// TwinCAT 3 PLC project MotionPractise
// ProgramVersion: 3.1.4023.0
// libraries:
//   Tc2_MC2, * (Beckhoff Automation GmbH)
//   Tc2_Standard, * (Beckhoff Automation GmbH)
//   Tc2_System, * (Beckhoff Automation GmbH)
//   Tc3_Module, * (Beckhoff Automation GmbH)
// project tree:
//   / PlcTask.TcTTO
//   POUs/AxisInterface/ Global_Axif_Const.TcGVL, Global_Axis_Interface.TcGVL, TE_AxisBasic_V2.TcPOU, TE_AxisInterface_type01.TcPOU
//   POUs/AxisInterface/Type/ Axis_Ctrl_gb.TcDUT, Axis_Status_gb.TcDUT, E_MotorDirection.TcDUT
//   POUs/AxisInterface/Type/Control/ E_AXIS_MODE.TcDUT, ST_AXIS_ADMINISTRATION.TcDUT, ST_AXIS_MODE_BITS.TcDUT, ST_AXIS_POSITION.TcDUT, ST_AXIS_SETUP_MODE.TcDUT, ST_AXIS_SYNCHRONISATION.TcDUT, ST_AXIS_TORQUE.TcDUT, ST_AXIS_VELOCITY.TcDUT, U_AXIS_MODE.TcDUT
//   POUs/AxisInterface/Type/Status/ ST_AXIS_ADMIN_STATUS.TcDUT, ST_AXIS_DIAGNOSIS.TcDUT, ST_AXIS_POS_STATUS.TcDUT, ST_AXIS_SETUP_MODE_STATUS.TcDUT, ST_AXIS_SYNC_STATUS.TcDUT, ST_AXIS_VEL_STATUS.TcDUT
//   POUs/ MAIN.TcPOU
// real-time tasks:
//   TASK PlcTask: cycle T#10ms, priority 20, ADS port 350
// motion (NC):
//   TASK NC-Task 1 SAF: cycle T#2ms, priority 4, ADS port 501
//   TASK NC-Task 1 SVB: cycle T#10ms, priority 8, ADS port 511
//   AXIS Axis 1 (id 1)
//     OtherSettings: AllowMotionCmdToSlave=true
//     encoder EncType=1
//     drive DrvType=5
//       Analog: TorqueSetpointScale=10, ScaleFactorActTorque=0.1
//     controller CtrType=1
//       CtrPara: PriorControlFactor=1
//         Observer: BandWidth=20
//   AXIS Axis 2 (id 2)
//     OtherSettings: AllowMotionCmdToSlave=true
//     encoder EncType=1
//     drive DrvType=5
//       Analog: TorqueSetpointScale=10, ScaleFactorActTorque=0.1
//     controller CtrType=1
//       CtrPara: PriorControlFactor=1
//         Observer: BandWidth=20
// variable links:
//   MotionPractise/MotionPractise Instance <-> NC-Task 1 SAF/Axes/Axis 1
//     PlcTask Inputs/Global_Axis_Interface.arAxisCtrl_gb[1].Admin.Axis.NcToPlc <-> Outputs/ToPlc
//     PlcTask Outputs/Global_Axis_Interface.arAxisCtrl_gb[1].Admin.Axis.PlcToNc <-> Inputs/FromPlc
//   MotionPractise/MotionPractise Instance <-> NC-Task 1 SAF/Axes/Axis 2
//     PlcTask Inputs/Global_Axis_Interface.arAxisCtrl_gb[2].Admin.Axis.NcToPlc <-> Outputs/ToPlc
//     PlcTask Outputs/Global_Axis_Interface.arAxisCtrl_gb[2].Admin.Axis.PlcToNc <-> Inputs/FromPlc

CONFIGURATION MotionPractise
    RESOURCE PLC ON TwinCAT3
        TASK PlcTask(INTERVAL := T#10ms, PRIORITY := 20);
        PROGRAM MAIN WITH PlcTask : MAIN;
    END_RESOURCE
END_CONFIGURATION

// ---- POUs/AxisInterface/Type/Axis_Ctrl_gb.TcDUT
TYPE
    Axis_Ctrl_gb :
    STRUCT
        Admin      : ST_AXIS_ADMINISTRATION;  // Administration of the Axis
        PosMode    : ST_AXIS_POSITION;        // Operating mode positioning (absolute, rel, additive)
        VelMode    : ST_AXIS_VELOCITY;        // Operation mode velocity control
        SyncMode   : ST_AXIS_SYNCHRONISATION; // Operation mode synchronisation(phase, vel and cam)
        TorqueMode : ST_AXIS_TORQUE;          // Operation mode / force control
        SetupMode  : ST_AXIS_SETUP_MODE;      // Jog / Homing functionality
    END_STRUCT
END_TYPE

// ---- POUs/AxisInterface/Type/Axis_Status_gb.TcDUT
TYPE
    Axis_Status_gb :
    STRUCT
        Admin     : ST_AXIS_ADMIN_STATUS;
        Diag      : ST_AXIS_DIAGNOSIS;
        PosMode   : ST_AXIS_POS_STATUS;
        VelMode   : ST_AXIS_VEL_STATUS;
        SyncMode  : ST_AXIS_SYNC_STATUS;
        SetupMode : ST_AXIS_SETUP_MODE_STATUS;
    END_STRUCT
END_TYPE

// ---- POUs/AxisInterface/Type/Control/E_AXIS_MODE.TcDUT
TYPE E_AXIS_MODE :
    (
        ModeAb             := 0,
        ModeAH             := 1,
        ModeHoming         := 2,
        ModePosAbs         := 4,
        ModePosRel         := 8,
        ModePosAdd         := 16,
        ModeVel            := 32,
        ModeSyncPhase      := 64,
        ModeSyncVel        := 128,
        ModeSyncCam        := 256,
        ModeSyncProfile    := 512,
        ModeTorque         := 1024,
        ModeFlexProfile    := 2048,
        ModeStopping       := 4096,
        ModeCoordinated    := 8192,
        ModeInterrupted    := 16384,
        ModeExternalFB     := 32768,
        ModeCyclicPosition := 65536,
        ModeCyclicVelocity := 131072,
        ModeCyclicTorque   := 262144
    ) UDINT;
END_TYPE

// ---- POUs/AxisInterface/Type/Control/ST_AXIS_ADMINISTRATION.TcDUT
TYPE ST_AXIS_ADMINISTRATION :
STRUCT
	//OpMode 
	Axis : AXIS_REF; // The reference to this Axis
	_OpMode : U_AXIS_MODE; // Selection of the operating mode
	StopDeceleration : LREAL; // Deceleration parameter used when an Axis executes a Stop. 
END_STRUCT
END_TYPE

// ---- POUs/AxisInterface/Type/Control/ST_AXIS_MODE_BITS.TcDUT
TYPE ST_AXIS_MODE_BITS :
STRUCT
        ModeAb             :BIT;
        ModeAH             :BIT;
        ModeHoming         :BIT;
        ModePosAbs         :BIT;
        ModePosRel         :BIT;
        ModePosAdd         :BIT;
        ModeVel            :BIT;
        ModeSyncPhase      :BIT;
        ModeSyncVel        :BIT;
        ModeSyncCam        :BIT;
        ModeSyncProfile    :BIT;
        ModeTorque         :BIT;
        ModeFlexProfile    :BIT;
        ModeStopping       :BIT;
        ModeCoordinated    :BIT;
        ModeInterrupted    :BIT;
        ModeExternalFB     :BIT;
        ModeCyclicPosition :BIT;
        ModeCyclicVelocity :BIT;
        ModeCyclicTorque   :BIT;
END_STRUCT
END_TYPE

// ---- POUs/AxisInterface/Type/Control/ST_AXIS_POSITION.TcDUT
TYPE ST_AXIS_POSITION :
STRUCT
END_STRUCT
END_TYPE

// ---- POUs/AxisInterface/Type/Control/ST_AXIS_SETUP_MODE.TcDUT
TYPE ST_AXIS_SETUP_MODE :
STRUCT
END_STRUCT
END_TYPE

// ---- POUs/AxisInterface/Type/Control/ST_AXIS_SYNCHRONISATION.TcDUT
TYPE ST_AXIS_SYNCHRONISATION :
STRUCT
END_STRUCT
END_TYPE

// ---- POUs/AxisInterface/Type/Control/ST_AXIS_TORQUE.TcDUT
TYPE ST_AXIS_TORQUE :
STRUCT
END_STRUCT
END_TYPE

// ---- POUs/AxisInterface/Type/Control/ST_AXIS_VELOCITY.TcDUT
TYPE ST_AXIS_VELOCITY :
STRUCT
END_STRUCT
END_TYPE

// ---- POUs/AxisInterface/Type/Control/U_AXIS_MODE.TcDUT
TYPE U_AXIS_MODE :
UNION
	en : E_AXIS_MODE;
	b: ST_AXIS_MODE_BITS;
END_UNION
END_TYPE

// ---- POUs/AxisInterface/Type/E_MotorDirection.TcDUT
TYPE E_MotorDirection :
(
	NoDirection := 0,
	OnlyPostive,
	OnlyNegative,
	Two_Way
)INT;
END_TYPE

// ---- POUs/AxisInterface/Type/Status/ST_AXIS_ADMIN_STATUS.TcDUT
TYPE ST_AXIS_ADMIN_STATUS :
    STRUCT
        _OpModeAck         :E_AXIS_MODE;
        ModeAb             :BIT;
        ModeAH             :BIT;
        ModeHoming         :BIT;
        ModePosAbs         :BIT;
        ModePosRel         :BIT;
        ModePosAdd         :BIT;
        ModeVel            :BIT;
        ModeSyncPhase      :BIT;
        ModeSyncVel        :BIT;
        ModeSyncCam        :BIT;
        ModeSyncProfile    :BIT;
        ModeTorque         :BIT;
        ModeFlexProfile    :BIT;
        ModeStopping       :BIT;
        ModeCoordinated    :BIT;
        ModeInterrupted    :BIT;
        ModeExternalFB     :BIT;
        ModeCyclicPosition :BIT;
        ModeCyclicVelocity :BIT;
        ModeCyclicTorque   :BIT;
        Active             :BOOL;
        CmdDone            :BOOL;
    END_STRUCT
END_TYPE

// ---- POUs/AxisInterface/Type/Status/ST_AXIS_DIAGNOSIS.TcDUT
TYPE ST_AXIS_DIAGNOSIS :
STRUCT
END_STRUCT
END_TYPE

// ---- POUs/AxisInterface/Type/Status/ST_AXIS_POS_STATUS.TcDUT
TYPE ST_AXIS_POS_STATUS :
STRUCT
END_STRUCT
END_TYPE

// ---- POUs/AxisInterface/Type/Status/ST_AXIS_SETUP_MODE_STATUS.TcDUT
TYPE ST_AXIS_SETUP_MODE_STATUS :
STRUCT
END_STRUCT
END_TYPE

// ---- POUs/AxisInterface/Type/Status/ST_AXIS_SYNC_STATUS.TcDUT
TYPE ST_AXIS_SYNC_STATUS :
STRUCT
END_STRUCT
END_TYPE

// ---- POUs/AxisInterface/Type/Status/ST_AXIS_VEL_STATUS.TcDUT
TYPE ST_AXIS_VEL_STATUS :
STRUCT
END_STRUCT
END_TYPE

// ---- POUs/AxisInterface/Global_Axif_Const.TcGVL
VAR_GLOBAL CONSTANT
	uiMAX_AXIS_INDEX : UINT := 40; // Maximum number of servos in the system.
	uiMAX_AXIS_NUMBER: UINT := 2; // Actual number of servos in the system.
END_VAR

// ---- POUs/AxisInterface/Global_Axis_Interface.TcGVL
VAR_GLOBAL
	arAxisCtrl_gb : ARRAY[1..uiMAX_AXIS_INDEX] OF Axis_Ctrl_gb;
	arAxisStutus_gb : ARRAY[1..uiMAX_AXIS_INDEX] OF Axis_Status_gb;
END_VAR

// ---- POUs/MAIN.TcPOU
PROGRAM MAIN
VAR
END_VAR

END_PROGRAM

// ---- POUs/AxisInterface/TE_AxisBasic_V2.TcPOU
FUNCTION_BLOCK TE_AxisBasic_V2
VAR_INPUT
END_VAR

VAR_OUTPUT
END_VAR

VAR
    PowerControl :MC_Power;
    bAxisEnable  :BOOL;
	{attribute 'no_copy'}
    AdminCtrl      :REFERENCE TO ST_AXIS_ADMINISTRATION;
	{attribute 'no_copy'}
    PosModeCtrl    :REFERENCE TO ST_AXIS_POSITION;
	{attribute 'no_copy'}
    VelModeCtrl    :REFERENCE TO ST_AXIS_VELOCITY;
	{attribute 'no_copy'}
    SyncModeCtrl   :REFERENCE TO ST_AXIS_SYNCHRONISATION;
	{attribute 'no_copy'}
    TorqueModeCtrl :REFERENCE TO ST_AXIS_TORQUE;
	{attribute 'no_copy'}
    SetupModeCtrl  :REFERENCE TO ST_AXIS_SETUP_MODE;
	{attribute 'no_copy'}
	AdminStatus : REFERENCE TO ST_AXIS_ADMIN_STATUS;
	{attribute 'no_copy'}
	DiagStatus : REFERENCE TO ST_AXIS_DIAGNOSIS;
	{attribute 'no_copy'}
	PosModeStatus : REFERENCE TO ST_AXIS_POS_STATUS;
	{attribute 'no_copy'}
	VelModeStatus : REFERENCE TO ST_AXIS_VEL_STATUS;
	{attribute 'no_copy'}
	SyncModeStatus: REFERENCE TO ST_AXIS_SYNC_STATUS;
	{attribute 'no_copy'}
	SetupModeStatus: REFERENCE TO ST_AXIS_SETUP_MODE_STATUS;
	ClearError: MC_Reset;
	bAxisStop: BOOL;
END_VAR


//=========================================//
// Cyclic update						   //
//=========================================//
A90_Cyclic();

ACTION A00_ModeAb:
// Check Reference available
IF NOT __ISVALIDREF(AdminCtrl) THEN
	RETURN;
END_IF

// Check Operation mode is ModeAb
IF AdminCtrl._OpMode.en <> ModeAb THEN
	RETURN;
END_IF

// Check Axis Servo OFF
IF NOT  AdminCtrl.Axis.Status.Disabled THEN
	AdminStatus.ModeAb := TRUE;
	AdminStatus._OpModeAck := ModeAb;
	AdminStatus.CmdDone := TRUE;
END_IF
END_ACTION

ACTION A01_ModeAH:
IF AdminCtrl._OpMode.en <> ModeAH THEN
	RETURN;
END_IF

IF AdminCtrl.Axis.Status.StandStill THEN
	AdminCtrl.Axis.Status.
END_IF
END_ACTION

ACTION A90_Cyclic:
PowerControl(Axis := AdminCtrl.Axis, Enable := bAxisEnable); // MC_Power
MC_Stop(Axis := AdminCtrl.Axis, Execute := bAxisStop, Deceleration := AdminCtrl.StopDeceleration);
MC_Jog(Axis := AdminCtrl.Axis);
ClearError(Axis := AdminCtrl.Axis); // MC_Reset
MC_Home(Axis := AdminCtrl.Axis);
MC_MoveAbsolute(Axis := AdminCtrl.Axis);
MC_MoveVelocity(Axis := AdminCtrl.Axis);
MC_Halt(Axis := AdminCtrl.Axis);
MC_MoveRelative(Axis := AdminCtrl.Axis);
MC_ReadAxisError(Axis := AdminCtrl.Axis);
MC_ReadActualPosition(Axis := AdminCtrl.Axis);
MC_ReadActualVelocity(Axis := AdminCtrl.Axis);
END_ACTION

METHOD M_GetOpMode : E_AXIS_MODE
VAR_INPUT
END_VAR
IF __ISVALIDREF(AdminStatus) THEN
	M_GetOpMode := AdminStatus._OpModeAck;
END_IF
END_METHOD

METHOD M_InitExtension
VAR_INPUT
	Index : UINT;
END_VAR
//=============================================================//
//Reference access											   //
//=============================================================//
AdminCtrl      REF= arAxisCtrl_gb[Index].Admin;
PosModeCtrl    REF= arAxisCtrl_gb[Index].PosMode;
VelModeCtrl    REF= arAxisCtrl_gb[Index].VelMode;
SyncModeCtrl   REF= arAxisCtrl_gb[Index].SyncMode;
TorqueModeCtrl REF= arAxisCtrl_gb[Index].TorqueMode;
SetupModeCtrl  REF= arAxisCtrl_gb[Index].SetupMode;

AdminStatus     REF= arAxisStutus_gb[Index].Admin;
DiagStatus      REF= arAxisStutus_gb[Index].Diag;
PosModeStatus   REF= arAxisStutus_gb[Index].PosMode;
VelModeStatus   REF= arAxisStutus_gb[Index].VelMode;
SyncModeStatus  REF= arAxisStutus_gb[Index].SyncMode;
SetupModeStatus REF= arAxisStutus_gb[Index].SetupMode;
END_METHOD

END_FUNCTION_BLOCK

// ---- POUs/AxisInterface/TE_AxisInterface_type01.TcPOU
PROGRAM TE_AxisInterface_type01
VAR_INPUT
    ClearError :BOOL;
END_VAR

VAR
    uiState :UINT := STATE_FIRST_INIT; // statemachine
    uiLoop  :UINT := 1;
    fbAxis  :ARRAY[1..uiMAX_AXIS_NUMBER] OF TE_AxisBasic_V2;
END_VAR

VAR CONSTANT
    STATE_FIRST_INIT :UINT := 0;
    STATE_WAIT_ERROR :UINT := 1;
    STATE_PRG_ERROR  :UINT := 9;
END_VAR

VAR_OUTPUT
    InitDone :BOOL;
    ERROR    :BOOL;
END_VAR

CASE uiState OF
    STATE_FIRST_INIT:
        // Add first cycle want to set or reset prog
        FOR uiLoop := 1 TO uiMAX_AXIS_NUMBER DO
            ;
        END_FOR

        InitDone := FALSE;
        uiState  := STATE_WAIT_ERROR;
    STATE_WAIT_ERROR:
        InitDone := TRUE;
    STATE_PRG_ERROR:
        IF ClearError THEN
            ERROR   := FALSE;
            uiState := STATE_WAIT_ERROR;
        END_IF
ELSE
    ERROR   := TRUE;
    uiState := STATE_PRG_ERROR;
END_CASE

IF InitDone THEN
	//============================================//
	// Reflash Axis Interface					  //
	//============================================//
	FOR uiLoop := 1 TO uiMAX_AXIS_NUMBER DO
		fbAxis[uiLoop].M_InitExtension(uiLoop);
		fbAxis[uiLoop]();
	END_FOR
END_IF

END_PROGRAM
